{attribute 'linkalways'} 
{attribute 'no_explicit_call' := 'This FB is a CLASS and must be accessed using methods or properties'}
{attribute 'enable_dynamic_creation'}
FUNCTION_BLOCK Node_F_VN_PointToPointDirection_TcVnPoint2_REAL EXTENDS VisionNode
VAR
    aPoint1 : _TcVnPoint2_REAL;
    aPoint2 : _TcVnPoint2_REAL;
    aDirection : _TcVnVector2_REAL;
    bNormalize : _BOOL(FALSE);
    hrPrev : _HRESULT(S_OK);
	hresult : _HRESULT(S_OK);
END_VAR

METHOD PUBLIC  Clone : I_Node
VAR
	pNode : POINTER TO Node_F_VN_PointToPointDirection_TcVnPoint2_REAL;
END_VAR
pNode := __NEW(Node_F_VN_PointToPointDirection_TcVnPoint2_REAL);
Clone := pNode^;
END_METHOD

METHOD FB_init : BOOL
VAR_INPUT
	bInitRetains : BOOL; // if TRUE, the retain variables are initialized (warm start / cold start)
	bInCopyCode : BOOL;  // if TRUE, the instance afterwards gets moved into the copy code (online change)
END_VAR
AddInput('aPoint1', aPoint1);
AddInput('aPoint2', aPoint2);
AddParameter('bNormalize', bNormalize);
AddInput('hrPrev', hrPrev);
AddOutput('aDirection', aDirection);
AddOutput('hresult',hresult);
END_METHOD

METHOD PROTECTED OnExecute
hresult.Value := F_VN_PointToPointDirection_TcVnPoint2_REAL(
    aPoint1 := aPoint1.Value,
    aPoint2 := aPoint2.Value,
    aDirection := aDirection.Value,
    bNormalize := bNormalize.Value,
	hrPrev:= hrPrev.Value);
END_METHOD

METHOD PUBLIC PreExecutionCheck
VAR_INPUT
	Check : I_PreExecutionChecks;
END_VAR
END_METHOD

END_FUNCTION_BLOCK

(* stored: Version 1.1.0.1, ProductVersion 3.1.4024.15
   POU Node_F_VN_PointToPointDirection_TcVnPoint2_REAL: Id {88434916-973a-0a60-2a2e-791348b283e4}, SpecialFunc None
   Folder Constructor: Id {fc7f66b8-240f-03ae-2107-4d27d8e14387}
   Method Clone: Id {1fc2d637-a1c2-01ab-3fa5-e7aa2cee3f0e}
   Method FB_init: Id {44da43b9-57e6-0c50-08a7-12c7b7ba5e40}
   Method OnExecute: Id {b73d4e77-8214-08ff-3f79-56865cd1661e}
   Method PreExecutionCheck: Id {4f2886d9-8730-05a8-0608-3384a7cb926c} *)
